(* Logix 5000 project; controller WWTP_SOLIDS_CLX vendor 1 type 14 code 54 rev 17.2; software revision 17.00; part 16 of 16 *)
(* WAS_StorageTk_ToSolidsTk01_Pump600, continued *)

ROUTINE Main   (* ladder *)
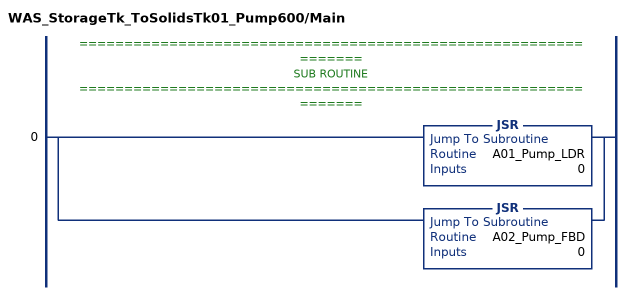
   // ===============================================================
   // SUB ROUTINE
   // ===============================================================
   0: [JSR(A01_Pump_LDR,0) ,JSR(A02_Pump_FBD,0) ];
END_ROUTINE
END_PROGRAM
